FUNCTION_BLOCK COUNTER
  {SET_ATTRIBUTE(OpcUa, DEVICE.SENSOR)}
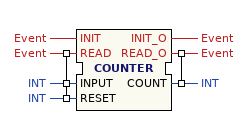
  EVENT_INPUT
    INIT;
    READ WITH INPUT, RESET;
  END_EVENT
  EVENT_OUTPUT
    INIT_O;
    READ_O WITH COUNT;
  END_EVENT
  VAR_INPUT
    INPUT : INT; {SET_ATTRIBUTE(OpcUa, Variable.RUN)}
    RESET : INT; {SET_ATTRIBUTE(OpcUa, Variable.RUN)}
  END_VAR
  VAR_OUTPUT
    COUNT : INT; {SET_ATTRIBUTE(OpcUa, Variable.RUN)}
  END_VAR
END_FUNCTION_BLOCK
